TYPE ERRORID : UINT; END_TYPE

(* stored: Version 1.1.0.1, ProductVersion 3.1.0.20
   DUT ERRORID: Id {6fda7034-3127-4f18-9536-cef88cd10ee9} *)
